SUBAPPLICATION Uebung_043 (* Scaling Function Block with limits Testing *)
  (* Standard: 61499-2; Description: Copyright (c) 2023 Meisterschulen am Ostbahnhof This program and the accompanying materials are made available under the terms of the Eclipse Public License 2.0 which is available at https://www.eclipse.org/legal/epl-2.0/ SPDX-License-Identifier: EPL-2.0 *)
  (* Version 1.0, 2023-10-23, Franz Höpfinger, Meisterschulen am Ostbahnhof, initial API and implementation and/or initial documentation *)
  PACKAGE Uebungen;
  IMPORT logiBUS::io::DI::logiBUS_DI::Input_I1;
  IMPORT logiBUS::io::DI::logiBUS_DI_Events::BUTTON_SINGLE_CLICK;
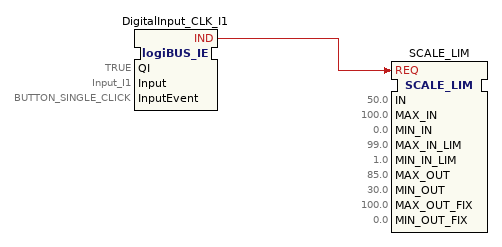
  FBS
    DigitalInput_CLK_I1 : logiBUS::io::DI::logiBUS_IE(QI := TRUE, Input := Input_I1, InputEvent := BUTTON_SINGLE_CLICK);
    SCALE_LIM : eclipse4diac::signalprocessing::SCALE_LIM(IN := 50.0, MAX_IN := 100.0, MIN_IN := 0.0, MAX_IN_LIM := 99.0, MIN_IN_LIM := 1.0, MAX_OUT := 85.0, MIN_OUT := 30.0, MAX_OUT_FIX := 100.0, MIN_OUT_FIX := 0.0);
  END_FBS
  EVENT_CONNECTIONS
    DigitalInput_CLK_I1.IND TO SCALE_LIM.REQ;
  END_CONNECTIONS
END_SUBAPPLICATION
